% RSLogix 500 project I2P-JOB23-ADAM BOCZKIEWICZ_BAK053.RSS, saved by version 10.00.00.00 %
PROJECT "ML04A"    % processor: Bul.1763 MicroLogix 1100 Series B %

PROGRAM FILES
  LAD 2   18 rungs

DATA FILES
  O0 OUTPUT  4 elements
  I1 INPUT  6 elements
  S2 STATUS  66 elements
  B3 BINARY  1 elements
  T4 TIMER  1 elements
  C5 COUNTER  2 elements
  R6 CONTROL  1 elements
  N7 INTEGER  1 elements
  F8 FLOAT  1 elements

LADDER 2
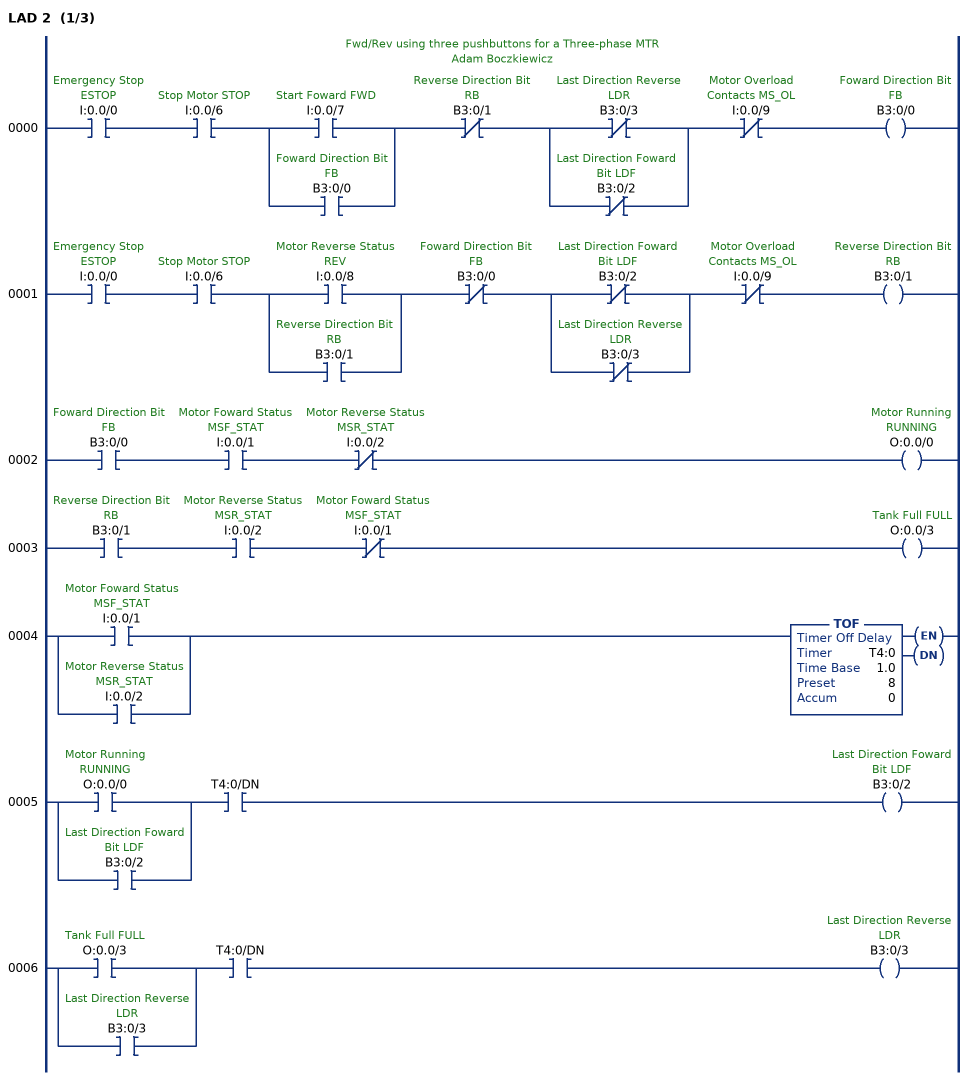
% Rung: 0 %
% Fwd/Rev using three pushbuttons for a Three-phase MTR
% Adam Boczkiewicz %
SOR XIC I:0.0/0 XIC I:0.0/6 BST XIC I:0.0/7 NXB XIC B3:0/0 BND XIO B3:0/1 BST XIO B3:0/3 NXB XIO B3:0/2 BND XIO I:0.0/9 OTE B3:0/0 EOR
%   I:0.0/0  ESTOP  "Emergency Stop" %
%   I:0.0/6  STOP  "Stop Motor" %
%   I:0.0/7  FWD  "Start Foward" %
%   B3:0/0  FB  "Foward Direction Bit" %
%   B3:0/1  RB  "Reverse Direction Bit" %
%   B3:0/3  LDR  "Last Direction Reverse" %
%   B3:0/2  LDF  "Last Direction Foward Bit" %
%   I:0.0/9  MS_OL  "Motor Overload Contacts" %
% Rung: 1 %
SOR XIC I:0.0/0 XIC I:0.0/6 BST XIC I:0.0/8 NXB XIC B3:0/1 BND XIO B3:0/0 BST XIO B3:0/2 NXB XIO B3:0/3 BND XIO I:0.0/9 OTE B3:0/1 EOR
%   I:0.0/0  ESTOP  "Emergency Stop" %
%   I:0.0/6  STOP  "Stop Motor" %
%   I:0.0/8  REV  "Motor Reverse Status" %
%   B3:0/1  RB  "Reverse Direction Bit" %
%   B3:0/0  FB  "Foward Direction Bit" %
%   B3:0/2  LDF  "Last Direction Foward Bit" %
%   B3:0/3  LDR  "Last Direction Reverse" %
%   I:0.0/9  MS_OL  "Motor Overload Contacts" %
% Rung: 2 %
SOR XIC B3:0/0 XIC I:0.0/1 XIO I:0.0/2 OTE O:0.0/0 EOR
%   B3:0/0  FB  "Foward Direction Bit" %
%   I:0.0/1  MSF_STAT  "Motor Foward Status" %
%   I:0.0/2  MSR_STAT  "Motor Reverse Status" %
%   O:0.0/0  RUNNING  "Motor Running" %
% Rung: 3 %
SOR XIC B3:0/1 XIC I:0.0/2 XIO I:0.0/1 OTE O:0.0/3 EOR
%   B3:0/1  RB  "Reverse Direction Bit" %
%   I:0.0/2  MSR_STAT  "Motor Reverse Status" %
%   I:0.0/1  MSF_STAT  "Motor Foward Status" %
%   O:0.0/3  FULL  "Tank Full" %
% Rung: 4 %
SOR BST XIC I:0.0/1 NXB XIC I:0.0/2 BND TOF T4:0 1.0 8 0 EOR
%   I:0.0/1  MSF_STAT  "Motor Foward Status" %
%   I:0.0/2  MSR_STAT  "Motor Reverse Status" %
% Rung: 5 %
SOR BST XIC O:0.0/0 NXB XIC B3:0/2 BND XIC T4:0/DN OTE B3:0/2 EOR
%   O:0.0/0  RUNNING  "Motor Running" %
%   B3:0/2  LDF  "Last Direction Foward Bit" %
% Rung: 6 %
SOR BST XIC O:0.0/3 NXB XIC B3:0/3 BND XIC T4:0/DN OTE B3:0/3 EOR
%   O:0.0/3  FULL  "Tank Full" %
%   B3:0/3  LDR  "Last Direction Reverse" %

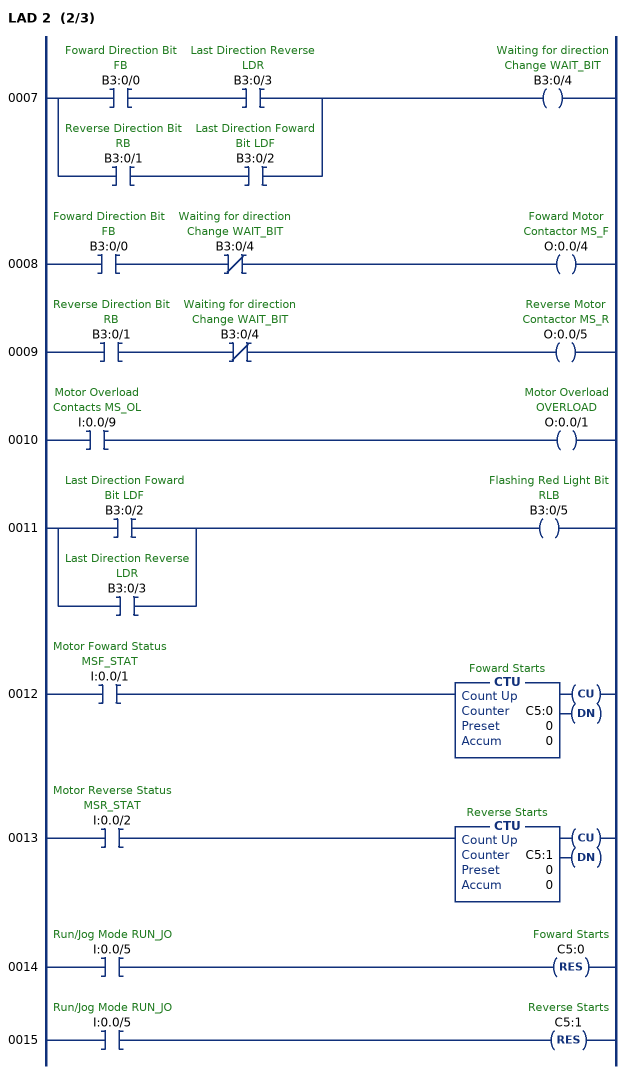
% Rung: 7 %
SOR BST XIC B3:0/0 XIC B3:0/3 NXB XIC B3:0/1 XIC B3:0/2 BND OTE B3:0/4 EOR
%   B3:0/0  FB  "Foward Direction Bit" %
%   B3:0/3  LDR  "Last Direction Reverse" %
%   B3:0/1  RB  "Reverse Direction Bit" %
%   B3:0/2  LDF  "Last Direction Foward Bit" %
%   B3:0/4  WAIT_BIT  "Waiting for direction Change" %
% Rung: 8 %
SOR XIC B3:0/0 XIO B3:0/4 OTE O:0.0/4 EOR
%   B3:0/0  FB  "Foward Direction Bit" %
%   B3:0/4  WAIT_BIT  "Waiting for direction Change" %
%   O:0.0/4  MS_F  "Foward Motor Contactor" %
% Rung: 9 %
SOR XIC B3:0/1 XIO B3:0/4 OTE O:0.0/5 EOR
%   B3:0/1  RB  "Reverse Direction Bit" %
%   B3:0/4  WAIT_BIT  "Waiting for direction Change" %
%   O:0.0/5  MS_R  "Reverse Motor Contactor" %
% Rung: 10 %
SOR XIC I:0.0/9 OTE O:0.0/1 EOR
%   I:0.0/9  MS_OL  "Motor Overload Contacts" %
%   O:0.0/1  OVERLOAD  "Motor Overload" %
% Rung: 11 %
SOR BST XIC B3:0/2 NXB XIC B3:0/3 BND OTE B3:0/5 EOR
%   B3:0/2  LDF  "Last Direction Foward Bit" %
%   B3:0/3  LDR  "Last Direction Reverse" %
%   B3:0/5  RLB  "Flashing Red Light Bit" %
% Rung: 12 %
SOR XIC I:0.0/1 CTU C5:0 0 0 EOR
%   I:0.0/1  MSF_STAT  "Motor Foward Status" %
%   C5:0  "Foward Starts" %
% Rung: 13 %
SOR XIC I:0.0/2 CTU C5:1 0 0 EOR
%   I:0.0/2  MSR_STAT  "Motor Reverse Status" %
%   C5:1  "Reverse Starts" %
% Rung: 14 %
SOR XIC I:0.0/5 RES C5:0 EOR
%   I:0.0/5  RUN_JO  "Run/Jog Mode" %
%   C5:0  "Foward Starts" %
% Rung: 15 %
SOR XIC I:0.0/5 RES C5:1 EOR
%   I:0.0/5  RUN_JO  "Run/Jog Mode" %
%   C5:1  "Reverse Starts" %

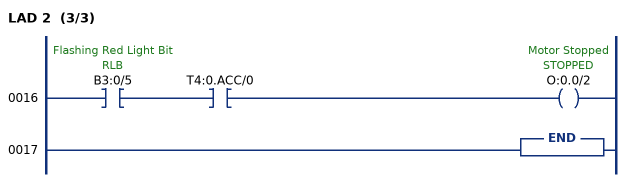
% Rung: 16 %
SOR XIC B3:0/5 XIC T4:0.ACC/0 OTE O:0.0/2 EOR
%   B3:0/5  RLB  "Flashing Red Light Bit" %
%   O:0.0/2  STOPPED  "Motor Stopped" %
% Rung: 17 %
SOR END EOR

OTHER DOCUMENTED ADDRESSES
  I:0.0/3  ON_MODE  "Mode: On Position"
  I:0.0/4  AUTO_MODE  "Mode: Auto Postion"
  JOG  
  MO  
  T4:0/TT  TT

DATA TABLE (non-zero values as saved)
DATA T4
% .PRE .ACC %
% T4:0 % 8 0
